{attribute 'GeneratedUsingTerminal: EP8309-0022-0021'}
{attribute addProperty BoxType "EP8309-0022-0021"}
{attribute addProperty Id "StatusAT %I*Status_72C27E804"}
{attribute addProperty CRC "2006162193"}
{attribute addProperty Size "4"}
TYPE PWM_Status_77939B11 EXTENDS InputBase_8311D824 :
STRUCT
	{attribute addProperty Name "Status"}
	Status AT %I* : Status_72C27E80;
END_STRUCT
END_TYPE

(* stored: Version 1.2.0.0, ProductVersion 3.1.4024.9
   DUT PWM_Status_77939B11: Id {40e71cc0-10ad-4cf3-8dab-29e0ccdfef23} *)
